# EPICS substitutions: fCCDApp/Db/user.substitutions
# Example substitutions file

file "db/dbExample1.db" {
    { user = "swilkins" }
}

file db/dbExample2.db {
    pattern { user, no, scan }
        { "swilkins", 1, "1 second" }
        { "swilkins", 2, "2 second" }
        { "swilkins", 3, "5 second" }
}
